// TIA Portal V19 export
TYPE "AnalogSens_HmiData"
   STRUCT
      PbPreset : Bool;   // Pulsante preset
      PresetValue : LReal;   // Valore di preset
      PresetFdback : LReal;   // Valore del sensore dopo il preset
   END_STRUCT;
END_TYPE
